(* CODESYS project tank1.project

Project tree, tasks and I/O mapping:
  Device : CODESYS Control Win V3 x64, 3S - Smart Software Solutions GmbH, version 3.5.16.20
    application Application
      libraries: Standard, 3.5.18.0 (System)
      task MainTask (cyclic, interval t#20ms, priority 1) calls Levels, Main, Simulate
      task VISU_TASK (cyclic, interval 100 ms, priority 31) calls VisuElems.Visu_Prg
      program Levels [FBD]
      program Main [SFC]: Init_level
      function block Process [SFC]
      global variables GVL
      program Simulate [ST]
      visualisation Visualization
  libraries: VisuSymbols, 4.4.0.0 (System)
  visualisation Visualization
  text list GlobalTextList
*)

// Device/Application/GVL
VAR_GLOBAL
	run: BOOL;
	level: REAL;
	empty: BOOL;
	full: BOOL;
	in_valve: BOOL;
	out_valve: BOOL;
	resistor: BOOL;
	temperature: REAL;
	hot: BOOL;
	stirrer: BOOL;
	counter: BOOL;
	i: INT:= 0;
END_VAR

VAR_GLOBAL
	step: INT;
END_VAR

// Device/Application/Levels
PROGRAM Levels
VAR
END_VAR

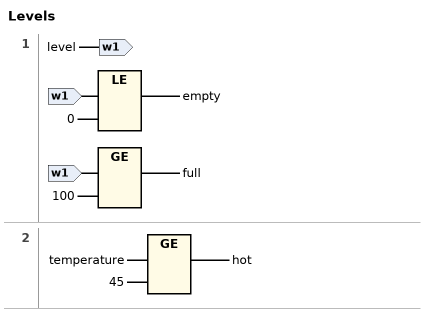
// NETWORK 1
empty := level <= 0;
full := level >= 100;

// NETWORK 2
hot := temperature >= 45;

END_PROGRAM

// Device/Application/Main
PROGRAM Main
VAR
	process: Process;
END_VAR

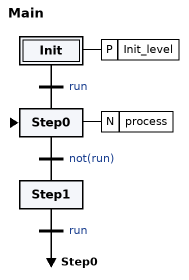
INITIAL_STEP Init:
    Init_level(P);
END_STEP
TRANSITION FROM Init TO Step0
    := run;
END_TRANSITION
STEP Step0:
    process(N);
END_STEP
TRANSITION FROM Step0 TO Step1
    := not(run);
END_TRANSITION
STEP Step1:
END_STEP
TRANSITION FROM Step1 TO Step0
    := run;
END_TRANSITION

ACTION Init_level:
level := 0;
END_ACTION

END_PROGRAM

// Device/Application/Process
FUNCTION_BLOCK Process

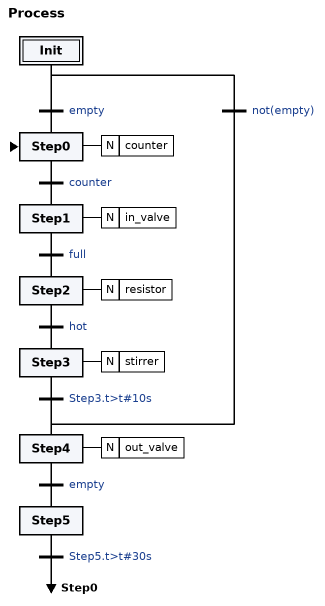
INITIAL_STEP Init:
END_STEP
TRANSITION FROM Init TO Step0
    := empty;
END_TRANSITION
STEP Step0:
    counter(N);
END_STEP
TRANSITION FROM Step0 TO Step1
    := counter;
END_TRANSITION
STEP Step1:
    in_valve(N);
END_STEP
TRANSITION FROM Step1 TO Step2
    := full;
END_TRANSITION
STEP Step2:
    resistor(N);
END_STEP
TRANSITION FROM Step2 TO Step3
    := hot;
END_TRANSITION
STEP Step3:
    stirrer(N);
END_STEP
TRANSITION FROM Step3 TO Step4
    := Step3.t>t#10s;
END_TRANSITION
TRANSITION FROM Init TO Step4
    := not(empty);
END_TRANSITION
STEP Step4:
    out_valve(N);
END_STEP
TRANSITION FROM Step4 TO Step5
    := empty;
END_TRANSITION
STEP Step5:
END_STEP
TRANSITION FROM Step5 TO Step0
    := Step5.t>t#30s;
END_TRANSITION

END_FUNCTION_BLOCK

// Device/Application/Simulate
PROGRAM Simulate

(* simulates level increase or decrease *)
(* according to valve status *)
IF (in_valve) THEN
   level := level + 0.2;
END_IF;
IF (out_valve) THEN
	IF level >= 0.2 THEN
   		level := level - 0.2;
	ELSE
		level := 0;
	END_IF
END_IF;

(* simulate temperature increase *)
(* according to resistor status *)
IF (resistor) THEN
	temperature := temperature + 0.1;
END_IF
IF (empty) THEN
	temperature := 21;
END_IF
IF (counter) THEN
	i := i + 1;
END_IF

END_PROGRAM

// /Visualization
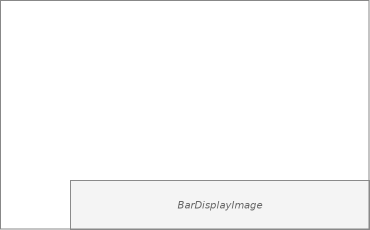
VISUALIZATION Visualization  // 370x230
    BarDisplayImage (70,180 300x50), value: temperature, style: BarDisplayImage-Gray, scale format: %.1f, scale 0..100
END_VISUALIZATION

// Device/Application/Visualization
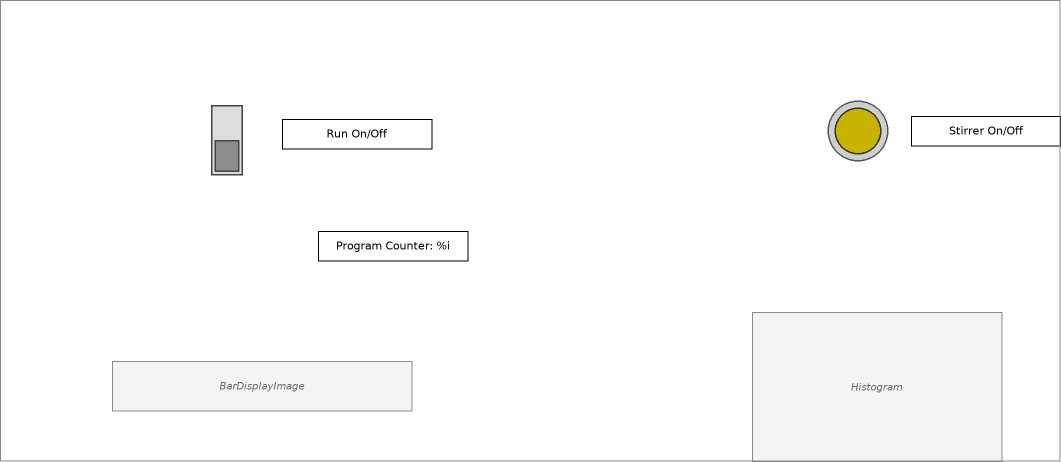
VISUALIZATION Visualization  // 1061x462
    DipSwitch (192,105 70x70), variable: run, behaviour: TOGGLE, style: Switch-DipSwitch-Gray
    Lamp1 (823,96 70x70), variable: stirrer, style: Lamp-Lamp1-Yellow
    BarDisplayImage (112,361 300x50), value: temperature, style: BarDisplayImage-Gray, scale format: %.1f, scale 0..100
        p518627256: Liquid Temperature
    Histogram (752,312 250x150), scale format: %.1f, scale 0..100
        p518627256: Liquid Levels
        p1518820177: level
        p102497268: level
    Rectangle (911,116 150x30), "Stirrer On/Off"
    Rectangle (282,119 150x30), "Run On/Off"
    Rectangle (318,231 150x30), "Program Counter: %i", text variable: i
END_VISUALIZATION
